(* CODESYS project Buffer Station - Barghash v3.0.project

Project tree, tasks and I/O mapping:
  Device : CODESYS Control Win V3, 3S - Smart Software Solutions GmbH, order no. 305021, version 3.5.11.30
    application Application
      libraries: Standard, * (System)
      task MainTask (cyclic, interval t#20ms, priority 1) calls PLC_PRG
      program PLC_PRG [LD]: A_Reset_Geral
      Symbols
*)

// Device/Application/PLC_PRG
PROGRAM PLC_PRG
VAR
	// --- Entradas (Mapear na image_6cef05.png) ---
	aux1				: BOOL; 
	FirstScan			: BOOL;
	xStart_Button       : BOOL; 
	xStop_Button        : BOOL; // NF
	xReset_Button       : BOOL; 
	P0_Home				: BOOL;
	P1_Alimentacao		: BOOL;
	P2_Rota_Metal		: BOOL;
	P3_Rota_Plastico	: BOOL;
	P4_Desvia_Plastico	: BOOL;
	P_Watchdog_Tempo	: BOOL;
	Remover_Plastico	: BOOL := TRUE;
	Remover_Metal		: BOOL := TRUE;

	
	Emitter				: BOOL;
	xConveyor_Motor		: INT;
	Pusher				: BOOL;
	Alarme_Erro_Discrepancia	: BOOL;
	
	
	S_Capacitivo		: BOOL;
	S_Indutivo			: BOOL;
	S_T3_Metal_Out		: BOOL;
	S_T5_Plastico_Out	: BOOL;
	T4_Wait_Pos			: TON;
	Tempo				: TIME;
	T_Max_Watchdog		: TON;
	Watchdog_Time		: TIME;
	trigReset      		: R_TRIG;

END_VAR
VAR // added by the converter: edge detectors and wires of the graphical bodies
    _w1, _w2, _w3, _w4, _w5, _w6, _w7, _w8 : BOOL;
END_VAR

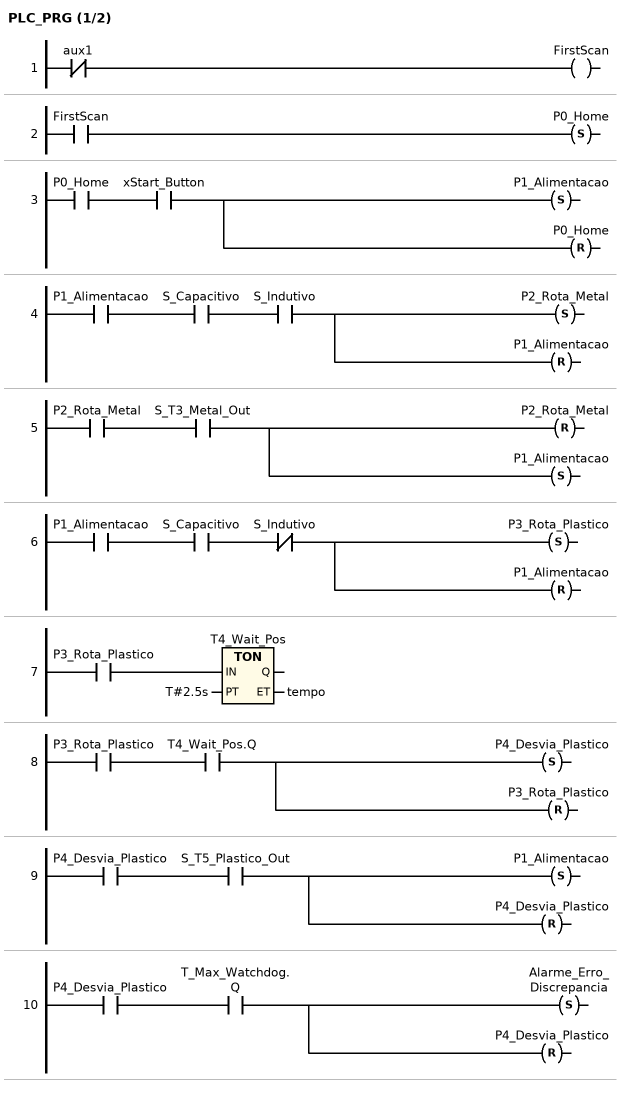
// NETWORK 1
FirstScan := NOT aux1;

// NETWORK 2
P0_Home S= FirstScan;

// NETWORK 3
_w1 := P0_Home AND xStart_Button;
P1_Alimentacao S= _w1;
P0_Home R= _w1;

// NETWORK 4
_w2 := P1_Alimentacao AND S_Capacitivo AND S_Indutivo;
P2_Rota_Metal S= _w2;
P1_Alimentacao R= _w2;

// NETWORK 5
_w3 := P2_Rota_Metal AND S_T3_Metal_Out;
P2_Rota_Metal R= _w3;
P1_Alimentacao S= _w3;

// NETWORK 6
_w4 := P1_Alimentacao AND S_Capacitivo AND NOT S_Indutivo;
P3_Rota_Plastico S= _w4;
P1_Alimentacao R= _w4;

// NETWORK 7
T4_Wait_Pos(IN := P3_Rota_Plastico, PT := T#2.5s, ET => tempo); // TON

// NETWORK 8
_w5 := P3_Rota_Plastico AND T4_Wait_Pos.Q;
P4_Desvia_Plastico S= _w5;
P3_Rota_Plastico R= _w5;

// NETWORK 9
_w6 := P4_Desvia_Plastico AND S_T5_Plastico_Out;
P1_Alimentacao S= _w6;
P4_Desvia_Plastico R= _w6;

// NETWORK 10
_w7 := P4_Desvia_Plastico AND T_Max_Watchdog.Q;
Alarme_Erro_Discrepancia S= _w7;
P4_Desvia_Plastico R= _w7;

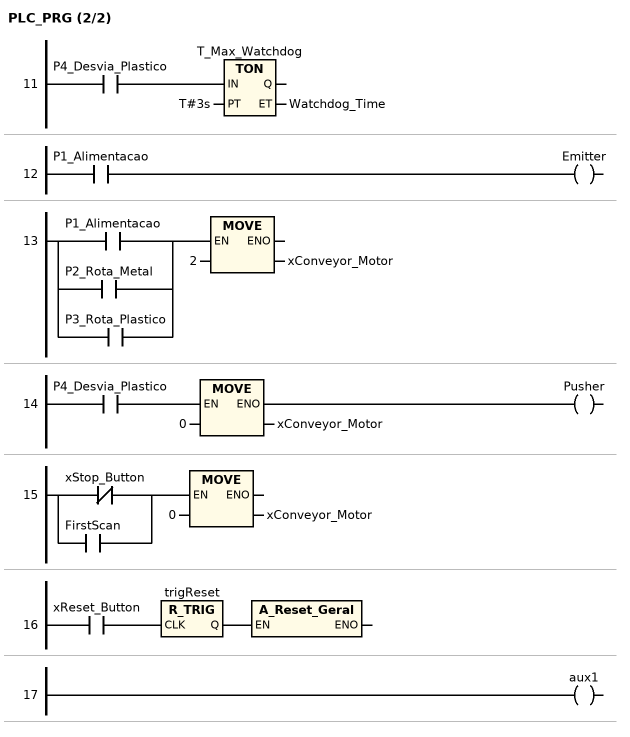
// NETWORK 11
T_Max_Watchdog(IN := P4_Desvia_Plastico, PT := T#3s, ET => Watchdog_Time); // TON

// NETWORK 12
Emitter := P1_Alimentacao;

// NETWORK 13
IF P1_Alimentacao OR P2_Rota_Metal OR P3_Rota_Plastico THEN xConveyor_Motor := 2; END_IF

// NETWORK 14
_w8 := P4_Desvia_Plastico;
IF _w8 THEN xConveyor_Motor := 0; END_IF
Pusher := _w8;

// NETWORK 15
IF NOT xStop_Button OR FirstScan THEN xConveyor_Motor := 0; END_IF

// NETWORK 16
trigReset(CLK := xReset_Button); // R_TRIG
IF trigReset.Q THEN A_Reset_Geral(); END_IF

// NETWORK 17
aux1 := TRUE;

ACTION A_Reset_Geral:
// --- ESTADO INICIAL E CONTROLE ---
aux1             := TRUE;    // Sistema inicia habilitado
FirstScan        := TRUE;    // Indica primeira varredura do CLP
xStart_Button    := FALSE;   // Limpa comando de partida
xStop_Button     := FALSE;   // Limpa comando de parada
xReset_Button    := FALSE;   // Limpa comando de reset
Remover_Plastico := TRUE;
Remover_Metal	 := TRUE;

// --- LUGARES DA REDE DE PETRI (MARCAÇÃO INICIAL) ---
P0_Home              := TRUE;   // Lugar inicial contendo o token
P1_Alimentacao       := FALSE;
P2_Rota_Metal        := FALSE;
P3_Rota_Plastico     := FALSE;
P4_Desvia_Plastico   := FALSE;

// --- SENSORES E SINAIS DE PROCESSO ---
S_Capacitivo         := FALSE;  // Sensor capacitivo sem detecção
S_Indutivo           := FALSE;  // Sensor indutivo sem detecção
P_Watchdog_Tempo     := FALSE;  // Watchdog sem indicação de falha

// --- SINAIS DE TRANSIÇÃO E FLAGS ---
S_T3_Metal_Out       := FALSE;  // Limpa memória da transição de metal
S_T5_Plastico_Out    := FALSE;  // Limpa memória da transição de plástico

// --- ATUADORES E SAÍDAS ---
Emitter                  := FALSE;  // Emissor desligado
Pusher                   := FALSE;  // Atuador recolhido
xConveyor_Motor          := 0;      // Esteira parada (INT)
Alarme_Erro_Discrepancia := FALSE;  // Sem alarme ativo

// --- TEMPORIZADORES E VARIÁVEIS DE TEMPO ---
Tempo               := T#0s;   // Zera variável de tempo
Watchdog_Time       := T#0s;   // Zera tempo do watchdog
T4_Wait_Pos(IN := FALSE);      // Reseta temporizador de posicionamento
T_Max_Watchdog(IN := FALSE);   // Reseta temporizador watchdog
END_ACTION

END_PROGRAM
